% RSLogix 500 project MATHS 1 Q_BAK008.RSS, saved by version 8.30.00.15 %
PROJECT "UNTITLED"    % processor: MicroLogix 1400 %

PROGRAM FILES
  LAD 2   2 rungs

DATA FILES
  O0 OUTPUT  6 elements
  I1 INPUT  8 elements
  S2 STATUS  66 elements
  B3 BINARY  1 elements
  T4 TIMER  1 elements
  C5 COUNTER  1 elements
  R6 CONTROL  1 elements
  N7 INTEGER  9 elements
  F8 FLOAT  1 elements

LADDER 2
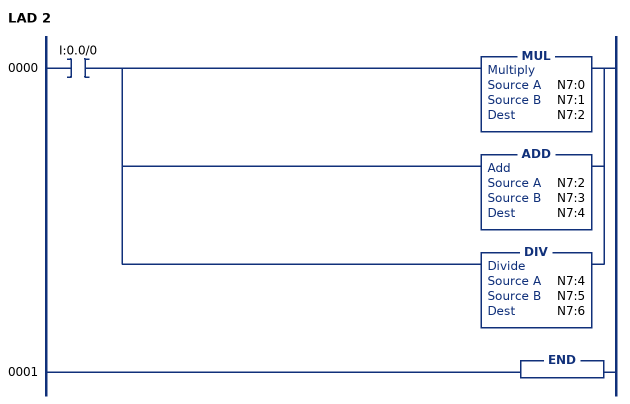
% Rung: 0 %
SOR XIC I:0.0/0 BST MUL N7:0 N7:1 N7:2 NXB BST ADD N7:2 N7:3 N7:4 NXB DIV N7:4 N7:5 N7:6 BND BND EOR
% Rung: 1 %
SOR END EOR

DATA TABLE (non-zero values as saved)
DATA N7
% N7:0 % 3 5 0 10 0 5 0 3 0
